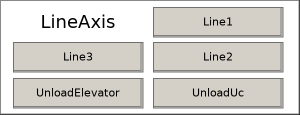
VISUALIZATION CtrlLine  // 300x115
    RoundedRectangle (0,0 300x115)
    Button (153,7 130x30), "Line1"
        OnMouseDown: execute { GVL.arrFbLine[E_Line.Line1].M_Jog(1); }
        OnMouseUp: execute { GVL.arrFbLine[E_Line.Line1].M_Jog(0); }
    Button (153,42 130x30), "Line2"
        OnMouseDown: execute { GVL.arrFbLine[E_Line.Line2].M_Jog(1); }
        OnMouseUp: execute { GVL.arrFbLine[E_Line.Line2].M_Jog(0); }
    Button (13,42 130x30), "Line3"
        OnMouseDown: execute { GVL.arrFbLine[E_Line.Line3].M_Jog(1); }
        OnMouseUp: execute { GVL.arrFbLine[E_Line.Line3].M_Jog(0); }
    Button (153,78 130x30), "UnloadUc"
        OnMouseDown: execute { GVL.arrFbLine[E_Line.UnloadUC].M_Jog(1); }
        OnMouseUp: execute { GVL.arrFbLine[E_Line.UnloadUC].M_Jog(0); }
    Button (13,78 130x30), "UnloadElevator"
        OnMouseDown: execute { GVL.arrFbLine[E_Line.UnloadElevator].M_Jog(1); }
        OnMouseUp: execute { GVL.arrFbLine[E_Line.UnloadElevator].M_Jog(0); }
    Label (13,7 130x30), "LineAxis"
END_VISUALIZATION

(* stored: Version 1.1.0.1, ProductVersion 3.1.4024.3
   Visu CtrlLine: Id {fe176b47-f187-4c6a-9336-8e4c0993602f} *)
